Universal Robots PolyScope program: Step Corner Around Up.urp

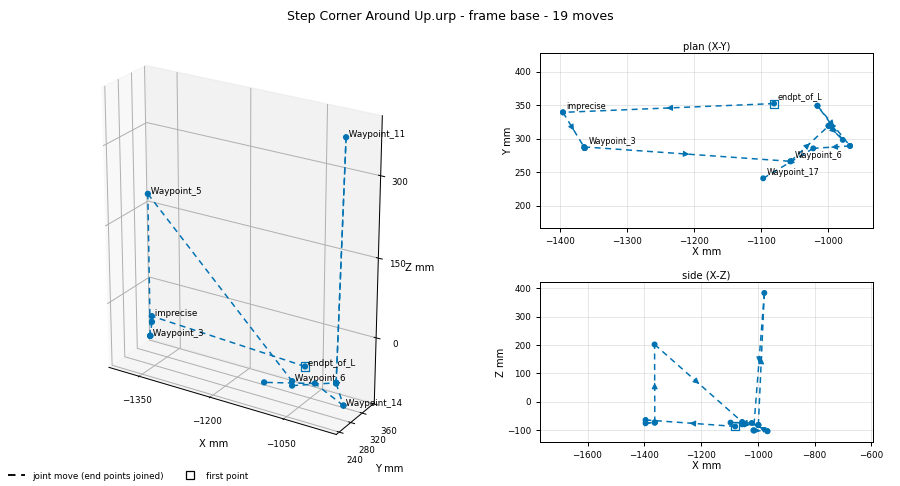
[picture p0: tool path of Step Corner Around Up.urp in frame base, 19 of 19 moves have a stored position in this frame; points joined in program order, loops and branches not executed]
Program Step Corner Around Up (installation=default directory=/programs createdIn=5.21.3 lastSavedIn=5.21.3 robotSerialNumber=20246801938)
Calibrated DH parameters: a=[-0.000071, -0.790281, -0.600694, 0.000061, -0.000039, 0]; d=[0.236272, 604.465945, 132.116513, -736.382239, 0.159268, 0.154005]; alpha=[1.570254, -0.000567, 0.000559, 1.571709, -1.56999, 0]; deltaTheta=[0, -0.409357, 7.293326, -0.600784, -0.000001, -0.000001]
InitVariablesNode
Robot Program (runOnlyOnce=false)
  Folder dummy points
    MoveJ speed 60 deg/s, acceleration 80 deg/s^2 (useActiveTCP=true optimoveEnabled=false optiMoveSpeed=0.3 optiMoveAcceleration=0.09) feature=Base
      Waypoint endpt_of_L: TCP in base x=-1080.054 y=352.633 z=-86.722 mm, rx=0.0341 ry=-0.0008 rz=-2.631 rad; joints [-41.761, 5.394, 77.547, 101.81, -19.08, -4.137] deg; TCP offset x=-9.5 y=-328 z=105.73 mm, rx=1.2092 ry=-1.2092 rz=1.2092 rad
    'left seam path'
    MoveJ speed 60 deg/s, acceleration 80 deg/s^2 (useActiveTCP=true optimoveEnabled=false optiMoveSpeed=0.3 optiMoveAcceleration=0.09) feature=Base
      Waypoint imprecise: TCP in base x=-1395.521 y=339.518 z=-63.924 mm, rx=0.0766 ry=-0.0347 rz=-2.5935 rad; joints [-31.708, 9.882, 49.427, 127.041, -27.073, -3.41] deg
      Waypoint Waypoint_2: TCP in base x=-1395.521 y=339.518 z=-75.451 mm, rx=0.0134 ry=-0.0524 rz=-2.5951 rad; joints [-31.054, 13.157, 42.809, 124.242, -27.702, 2.062] deg
      Waypoint Waypoint_3: TCP in base x=-1363.088 y=286.142 z=-72.943 mm, rx=0.0134 ry=-0.0524 rz=-2.5951 rad; joints [-29.664, 10.584, 50.73, 118.887, -29.093, 2.067] deg
      Waypoint Waypoint_1: TCP in base x=-1363.088 y=286.142 z=-72.943 mm, rx=0.2468 ry=-0.8856 rz=-2.4622 rad; joints [-24.351, 1.577, 73.674, 104.923, -34.409, 39.337] deg
      Waypoint Waypoint_4: TCP in base x=-1363.088 y=286.142 z=-72.943 mm, rx=0.5578 ry=-1.9956 rz=-1.8429 rad; joints [-20.064, -17.726, 96.684, 101.187, -38.706, 94.353] deg
      Waypoint Waypoint_5: TCP in base x=-1363.854 y=287.864 z=202.008 mm, rx=0.5349 ry=-1.9137 rz=-1.912 rad; joints [-20.125, -34.009, 104.192, 109.948, -38.652, 89.867] deg
    'right seam path'
    'must be closer'
    MoveJ speed 60 deg/s, acceleration 80 deg/s^2 (useActiveTCP=true optimoveEnabled=false optiMoveSpeed=0.3 optiMoveAcceleration=0.09) feature=Base
      Waypoint Waypoint_6: TCP in base x=-1055.377 y=266.316 z=-70.866 mm, rx=-0.0014 ry=0.0721 rz=-0.8224 rad; joints [-28.641, -7.044, 57.859, -54.616, -71.444, -180.462] deg
      Waypoint Waypoint_7: TCP in base x=-1055.377 y=266.316 z=-79.466 mm, rx=-0.0014 ry=0.0721 rz=-0.8224 rad; joints [-28.641, -6.518, 57.428, -54.711, -71.445, -180.462] deg
      Waypoint Waypoint_8: TCP in base x=-998.404 y=319.289 z=-81.739 mm, rx=-0.0014 ry=0.0721 rz=-0.8224 rad; joints [-31.903, -7.966, 61.956, -57.726, -74.698, -180.684] deg
      Waypoint Waypoint_9: TCP in base x=-998.404 y=319.289 z=-81.739 mm, rx=0.8845 ry=-0.3199 rz=-0.7932 rad; joints [-44.267, -18.687, 78.05, -62.97, -87.031, -127.542] deg
      Waypoint Waypoint_10: TCP in base x=-998.404 y=319.289 z=-81.739 mm, rx=1.4961 ry=-0.5974 rz=-0.6932 rad; joints [-47.849, -30.817, 85.526, -58.311, -90.6, -90.194] deg
      Waypoint Waypoint_11: TCP in base x=-977.341 y=298.379 z=383.404 mm, rx=1.4961 ry=-0.5974 rz=-0.6932 rad; joints [-47.912, -53.656, 85.268, -35.215, -90.659, -90.222] deg
    'under L path for closer'
    MoveJ speed 60 deg/s, acceleration 80 deg/s^2 (useActiveTCP=true optimoveEnabled=false optiMoveSpeed=0.3 optiMoveAcceleration=0.09) feature=Base
      'major problems regarding self collisions'
      Waypoint Waypoint_12: TCP in base x=-1015.127 y=349.357 z=-100.768 mm, rx=-0.0475 ry=0.0317 rz=-2.8842 rad; joints [-42.009, 6.908, 81.621, 88.667, -33.318, 0.794] deg
      Waypoint Waypoint_13: TCP in base x=-1015.127 y=349.357 z=-100.768 mm, rx=-0.0357 ry=0.0368 rz=-2.4594 rad; joints [-44.126, 7.34, 72.677, 93.591, -6.886, 4.286] deg
      Waypoint Waypoint_14: TCP in base x=-966.444 y=289.339 z=-103.526 mm, rx=-0.0357 ry=0.0368 rz=-2.4594 rad; joints [-43.532, 6.909, 79.202, 88.021, -7.474, 3.756] deg
      Waypoint Waypoint_15: TCP in base x=-966.444 y=289.339 z=-103.526 mm, rx=-0.0528 ry=0.0288 rz=-3.0604 rad; joints [-39.057, 7.474, 89.076, 80.978, -46.365, 0.452] deg
      Waypoint Waypoint_16: TCP in base x=-1021.437 y=285.676 z=-74.593 mm, rx=0.0494 ry=-0.0045 rz=2.303 rad; joints [-20.58, 5.315, 85.968, 86.294, -117.473, -0.511] deg
      Waypoint Waypoint_17: TCP in base x=-1096.236 y=240.938 z=-73.253 mm, rx=0.0496 ry=-0.0048 rz=2.3122 rad; joints [-16.366, 5.351, 80.35, 91.765, -121.158, -0.718] deg
